SYSTEM FLASHER_TESTRF (* Test FLASHER4 with Remote Frame *)
  (* Standard: 61499-1 *)
  (* Version 0.1, 2007-11-07, JHC, Holobloc Inc, RE-derived from FLASHER_TESTD. *)
  (* Version 0.0, 2006-10-26, JHC, Holobloc Inc, Derived from FLASHER_TESTD. *)
  DEVICE CTL_PANEL : FRAME_DEVICE(BOUNDS := [50,100,125,125], GRID := [1,1])
    RESOURCE RES1 : PANEL_RESOURCE
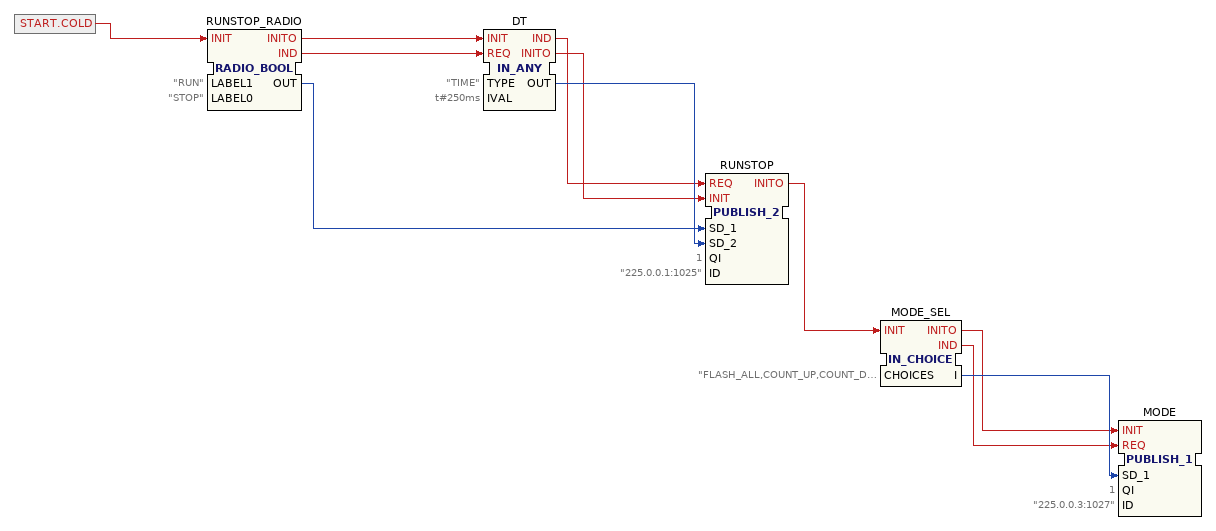
      FBS
        RUNSTOP_RADIO : RADIO_BOOL(LABEL1 := "RUN", LABEL0 := "STOP");
        MODE_SEL : IN_CHOICE(CHOICES := "FLASH_ALL,COUNT_UP,COUNT_DOWN,CHASE_UP,CHASE_DOWN");
        DT : IN_ANY(TYPE := "TIME", IVAL := t#250ms);
        RUNSTOP : PUBLISH_2(QI := 1, ID := "225.0.0.1:1025");
        MODE : PUBLISH_1(QI := 1, ID := "225.0.0.3:1027");
      END_FBS
      EVENT_CONNECTIONS
        START.COLD TO RUNSTOP_RADIO.INIT;
        RUNSTOP_RADIO.INITO TO DT.INIT;
        RUNSTOP_RADIO.IND TO DT.REQ;
        DT.IND TO RUNSTOP.REQ;
        DT.INITO TO RUNSTOP.INIT;
        RUNSTOP.INITO TO MODE_SEL.INIT;
        MODE_SEL.INITO TO MODE.INIT;
        MODE_SEL.IND TO MODE.REQ;
      END_CONNECTIONS
      DATA_CONNECTIONS
        RUNSTOP_RADIO.OUT TO RUNSTOP.SD_1;
        DT.OUT TO RUNSTOP.SD_2;
        MODE_SEL.I TO MODE.SD_1;
      END_CONNECTIONS
    END_RESOURCE
  END_DEVICE
  DEVICE FLASHER : RMT_FRAME(GRID := [1,1], BOUNDS := [175,100,225,75])
    RESOURCE RES1 : PANEL_RESOURCE
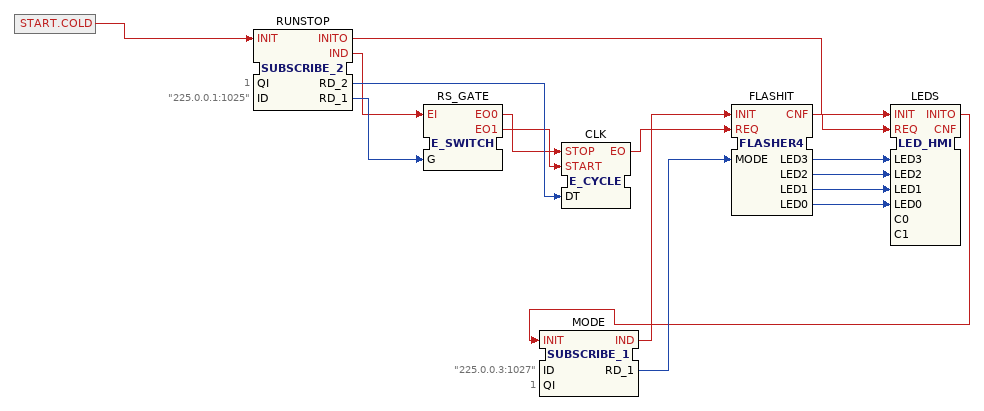
      FBS
        CLK : E_CYCLE;
        FLASHIT : FLASHER4;
        LEDS : LED_HMI;
        RUNSTOP : SUBSCRIBE_2(QI := 1, ID := "225.0.0.1:1025");
        RS_GATE : E_SWITCH;
        MODE : SUBSCRIBE_1(ID := "225.0.0.3:1027", QI := 1);
      END_FBS
      EVENT_CONNECTIONS
        CLK.EO TO FLASHIT.REQ;
        FLASHIT.CNF TO LEDS.REQ;
        START.COLD TO RUNSTOP.INIT;
        RUNSTOP.INITO TO LEDS.INIT;
        RUNSTOP.IND TO RS_GATE.EI;
        MODE.IND TO FLASHIT.INIT;
        LEDS.INITO TO MODE.INIT;
        RS_GATE.EO0 TO CLK.STOP;
        RS_GATE.EO1 TO CLK.START;
      END_CONNECTIONS
      DATA_CONNECTIONS
        FLASHIT.LED3 TO LEDS.LED3;
        FLASHIT.LED2 TO LEDS.LED2;
        FLASHIT.LED1 TO LEDS.LED1;
        FLASHIT.LED0 TO LEDS.LED0;
        RUNSTOP.RD_2 TO CLK.DT;
        RUNSTOP.RD_1 TO RS_GATE.G;
        MODE.RD_1 TO FLASHIT.MODE;
      END_CONNECTIONS
    END_RESOURCE
  END_DEVICE
END_SYSTEM
